// TIA Portal V17 export
// export: Created 2025-03-05T08:02:29.6923489Z, ExportSetting WithDefaults, DisplayName Totally Integrated Automation Portal, DisplayVersion V17 Update 8, DisplayName TIA Portal Openness, DisplayVersion V17 Update 8, DisplayName TIA Portal Version Control Interface, DisplayVersion V17, DisplayName SINAMICS Startdrive Advanced, DisplayVersion V17 SP2, DisplayName SINAMICS Startdrive G110M, G120, G120C, G120D, G120P, G115D, DisplayVersion V17 SP2, DisplayName SINAMICS Startdrive G130, G150, S120, S150, SINAMICS MV, S210, DisplayVersion V17 SP2, DisplayName STEP 7 Professional, DisplayVersion V17 Update 8, DisplayName SINUMERIK ONE STEP 7 Toolbox, DisplayVersion V17 Update 12, DisplayName SINUMERIK 840D sl STEP 7 Toolbox, DisplayVersion V17 Update 12, DisplayName STEP 7 Safety, DisplayVersion V17 Update 6, DisplayName WinCC Advanced, DisplayVersion V17 Update 8
TYPE "POWDER FEEDER GENERAL"
// stored: IsFailsafeCompliant false
   STRUCT
      "START GENERAL CONDITIONS" : Bool;   // Start General Conditions
      "START INITIAL CONDITIONS" : Bool;   // Start Initial Conditions
      "START MANUAL REQUEST" : Bool;   // Start Manual Request
      "START AUTO REQUEST" : Bool;   // Start Auto Request
      "START GLOBAL REQUEST" : Bool;   // Start Global Request
      "START COMMAND" : Bool;   // Start Command
      START : Bool;   // Start
      "FEEDBACK ON" : Bool;   // Feedback On
      "STOP GENERAL CONDITIONS" : Bool;   // Stop General Conditions
      "STOP INITIAL CONDITIONS" : Bool;   // Stop Initial Conditions
      "STOP MANUAL REQUEST" : Bool;   // Stop Manual Request
      "STOP AUTO REQUEST" : Bool;   // Stop Auto Request
      "STOP GLOBAL REQUEST" : Bool;   // Stop Global Request
      "STOP COMMAND" : Bool;   // Stop Command
      STOP : Bool;   // Stop
      "FEEDBACK OFF" : Bool;   // Feedback Off
      "FEEDBACK ON AUX FOR HMI" : Bool;   // Feedback On Aux for HMI
      "CG FEEDFUN DISABLED LINE 1" : Bool;   // CG Feedfun Disabled Line 1
      "CG READY START LINE 1" : Bool;   // CG Ready Start Line 1
      "CG WAIT TO ESTABLISH LINE 1" : Bool;   // CG Wait To Establish Line 1
      "FEEDFUNC READY START LINE 1" : Bool;   // Feedfunc Ready Start Line 1
      "FEEDFUN RUNNING LINE 1" : Bool;   // Feedfun Running Line 1
      "FEEDFUN WAIT TO ZERO LINE 1" : Bool;   // Feedfun Wait To Zero Line 1
      "CG FEEDFUN DISABLED LINE 2" : Bool;   // CG Feedfun Disabled Line 2
      "CG READY START LINE 2" : Bool;   // CG Ready Start Line 2
      "CG WAIT TO ESTABLISH LINE 2" : Bool;   // CG Wait To Establish Line 2
      "FEEDFUNC READY START LINE 2" : Bool;   // Feedfunc Ready Start Line 2
      "FEEDFUN RUNNING LINE 2" : Bool;   // Feedfun Running Line 2
      "FEEDFUN WAIT TO ZERO LINE 2" : Bool;   // Feedfun Wait To Zero Line 2
      "Mixer Fault" : Bool;   // Mixer Fault
      "Pressure Low Fault" : Bool;   // Pressure Low Fault
      "Gasflow Fault" : Bool;   // Gasflow Fault
      "Discflow Fault" : Bool;   // Discflow Fault
      "FEEDER PROFINET MODE ACTIVE" : Bool;   // Feeder Profinet Mode Active
      "FEEDER LINE 1 NOT READY FAULT" : Bool;   // Feeder Line 1 Not Ready Fault
      "FEEDER LINE 2 NOT READY FAULT" : Bool;   // Feeder Line 2 Not Ready Fault
      "FEEDER PROFINET MODE ACTIVE FAULT" : Bool;
      "Powder Line Clogged Line 1 Fault" : Bool;   // Powder Line Clogged Line 1 Fault
      "Powder Line Clogged Line 2 Fault" : Bool;   // Powder Line Clogged Line 2 Fault
      "Gas Flow Below Low Limit Line 1 Fault" : Bool;   // Gas Flow Below Low Limit Line 1 Fault
      "Gas Flow Below Low Limit Line 2 Fault" : Bool;   // Gas Flow Below Low Limit Line 2 Fault
      "Disk Speed Below Low Limit Line 1 Fault" : Bool;   // Disk Speed Below Low Limit Line 1 Fault
      "Disk Speed Below Low Limit Line 2 Fault" : Bool;   // Disk Speed Below Low Limit Line 2 Fault
      "Stirrer Speed Below Low Limit Line 1 Fault" : Bool;   // Stirrer Speed Below Low Limit Line 1 Fault
      "Stirrer Speed Below Low Limit Line 2 Fault" : Bool;   // Stirrer Speed Below Low Limit Line 2 Fault
      "Gas Flow Above High Limit Line 1 Fault" : Bool;   // Gas Flow Above High Limit Line 1 Fault
      "Gas Flow Above High Limit Line 2 Fault" : Bool;   // Gas Flow Above High Limit Line 2 Fault
      "Disk Speed Above High Limit Line 1 Fault" : Bool;   // Disk Speed Above High Limit Line 1 Fault
      "Disk Speed Above High Limit Line 2 Fault" : Bool;   // Disk Speed Above High Limit Line 2 Fault
      "Stirrer Speed Above High Limit Line 1 Fault" : Bool;   // Stirrer Speed Above High Limit Line 1 Fault
      "Stirrer Speed Above High Limit Line 2 Fault" : Bool;   // Stirrer Speed Above High Limit Line 2 Fault
      "Hopper Temperature Above High Limit Line 1 Fault" : Bool;   // Hopper Temperature Above High Limit Line 1 Fault
      "Hopper Temperature Above High Limit Line 2 Fault" : Bool;   // Hopper Temperature Above High Limit Line 2 Fault
      "Carrier Gas Inlet Pressure Too Low Line 1 Fault" : Bool;   // Carrier Gas Inlet Pressure Too Low Line 1 Fault
      "Carrier Gas Inlet Pressure Too Low Line 2 Fault" : Bool;   // Carrier Gas Inlet Pressure Too Low Line 2 Fault
      "Disk Motor Plugged In And Ready Line 1 Fault" : Bool;   // Disk Motor Plugged In And Ready Line 1 Fault
      "Disk Motor Plugged In And Ready Line 2 Fault" : Bool;   // Disk Motor Plugged In And Ready Line 2 Fault
      "Stirrer Plugged In And Ready Line 1 Fault" : Bool;   // Stirrer Plugged In And Ready Line 1 Fault
      "Stirrer Plugged In And Ready Line 2 Fault" : Bool;   // Stirrer Plugged In And Ready Line 2 Fault
      "Communication Running Line 1 Fault" : Bool;   // Communication Running Line 1 Fault
      "Communication Running Line 2 Fault" : Bool;   // Communication Running Line 2 Fault
      "Gas Flow Line 1 Under Warning" : Bool;   // Gas Flow Line 1 Under Warning
      "Gas Flow Line 2 Under Warning" : Bool;   // Gas Flow Line 2 Under Warning
      "Disk Speed Line 1 Under Warning" : Bool;   // Disk Speed Line 1 Under Warning
      "Disk Speed Line 2 Under Warning" : Bool;   // Disk Speed Line 2 Under Warning
      "Stirrer Speed Line 1 Under Warning" : Bool;   // Stirrer Speed Line 1 Under Warning
      "Stirrer Speed Line 2 Under Warning" : Bool;   // Stirrer Speed Line 2 Under Warning
      "Gas Flow Line 1 Over Warning" : Bool;   // Gas Flow Line 1 Over Warning
      "Gas Flow Line 2 Over Waning" : Bool;   // Gas Flow Line 2 Over Waning
      "Disk Speed Line 1 Over Warning" : Bool;   // Disk Speed Line 1 Over Warning
      "Disk Speed Line 2 Over Warning" : Bool;   // Disk Speed Line 2 Over Warning
      "Stirrer Speed Line 1 Over Warning" : Bool;   // Stirrer Speed Line 1 Over Warning
      "Stirrer Speed Line 2 Over Warning" : Bool;   // Stirrer Speed Line 2 Over Warning
      "Feeding Mode Gravimetric Line 1 Selected Warning" : Bool;   // Feeding Mode Gravimetric Line 1 Selected Warning
      "Feeding Mode Gravimetric Line 2 Selected Warning" : Bool;   // Feeding Mode Gravimetric Line 2 Selected Warning
      "CARRIER GAS IS RUNNING LINE 1" : Bool;   // Carrier Gas Is Running Line 1
      "CARRIER GAS IS OFFLINE 1" : Bool;   // Carrier Gas Is Off Line 1
      "CARRIER GAS IS RUNNING LINE 2" : Bool;   // Carrier Gas Is Running Line 2
      "CARRIER GAS IS OFFLINE 2" : Bool;   // Carrier Gas Is Off Line 2
      "Start General Conditions Help" : Bool;   // Start General Conditions Help
      "Start Initial Conditions Help" : Bool;   // Start Initial Conditions Help
      "Stop General Conditions Help" : Bool;   // Stop General Conditions Help
      "Stop Initial Conditions Help" : Bool;   // Stop Initial Conditions Help
      Fault : Bool;   // Fault
      "HMI Start" : Bool;   // HMI Start
      "HMI Stop" : Bool;   // HMI Stop
      "HMI Turned On" : Bool;   // HMI Turned On
      "HMI Turned Off" : Bool;   // HMI Turned Off
      "HMI Turning On" : Bool;   // HMI Turning On
      "HMI Turning Off" : Bool;   // HMI Turning Off
      "HMI Start Conditions" : Bool;   // HMI Start Conditions
      "HMI Stop Conditions" : Bool;   // HMI Stop Conditions
      "HMI Select G/Min Mode" : Bool;   // HMI Select G/Min Mode
      "HMI Turn On Powder Switch Nozzle" : Bool;   // HMI Turn On Powder Switch Nozzle
      "HMI Turn Off Powder Switch Nozzle" : Bool;   // HMI Turn Off Powder Switch Nozzle
      "HMI Switch On Profinet" : Bool;   // HMI Switch On Profinet
      "HMI Switch Off Profinet" : Bool;   // HMI Switch Off Profinet
      "HMI Set Temporal Disc RPMS" : Bool;   // HMI Set Temporal Disc RPMS
      "HMI Set Temporal Hopper Feedrate" : Bool;   // HMI Set Temporal Hopper Feedrate
      "HMI Set Temporal Gasflow" : Bool;   // HMI Set Temporal Gasflow
      "HMI Set Temporal Mixer" : Bool;   // HMI Set Temporal Mixer
      "HMI Actual Values Disc RPMS" : Bool;   // HMI Actual Values Disc RPMS
      "HMI Actual Values Hopper Feedrate" : Bool;   // HMI Actual Values Hopper Feedrate
      "HMI Actual Values Gasflow" : Bool;   // HMI Actual Values Gasflow
   END_STRUCT;
END_TYPE
